Omron CX-Programmer project NewProject (CX-Programmer 9.75)

# PLC parkir: CP1E N20

## Global symbols (name address type ; comment)
0.00 BOOL  ; MULAI
0.01 BOOL  ; STOP
0.02 BOOL  ; SENSOR MASUK
0.03 BOOL  ; SENSOR KELUAR
0.04 BOOL  ; RESET
100.00 BOOL  ; Portal Masuk
100.01 BOOL  ; Portal Keluar
100.02 BOOL  ; SPACE
100.03 BOOL  ; FULL
100.04 BOOL  ; FULL
10.00 BOOL  ; Relay
C2 CHANNEL  ; CNTR
T000 BOOL  ; TIMER
T001 BOOL  ; TIMER

## Program NewProgram1 (cyclic task 0)

### Section Section1

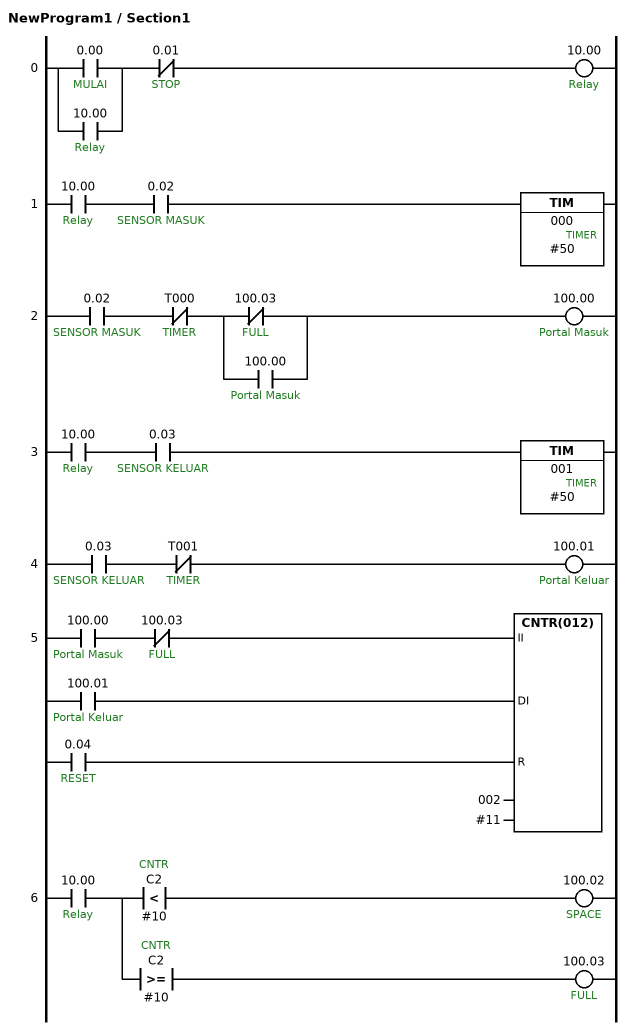
; rung 0
LD 0.00  ; MULAI
OR 10.00  ; Relay
ANDNOT 0.01  ; STOP
OUT 10.00  ; Relay
; rung 1
LD 10.00  ; Relay
AND 0.02  ; SENSOR MASUK
TIM 000 #50  ; TIMER
; rung 2
LD 0.02  ; SENSOR MASUK
ANDNOT T000  ; TIMER
LDNOT 100.03  ; FULL
OR 100.00  ; Portal Masuk
ANDLD
OUT 100.00  ; Portal Masuk
; rung 3
LD 10.00  ; Relay
AND 0.03  ; SENSOR KELUAR
TIM 001 #50  ; TIMER
; rung 4
LD 0.03  ; SENSOR KELUAR
ANDNOT T001  ; TIMER
OUT 100.01  ; Portal Keluar
; rung 5
LD 100.00  ; Portal Masuk
ANDNOT 100.03  ; FULL
LD 100.01  ; Portal Keluar
LD 0.04  ; RESET
CNTR(012) 002 #11
; rung 6
LD 10.00  ; Relay
OUT TR0
AND<(310) C2 #10  ; CNTR
OUT 100.02  ; SPACE
LD TR0
AND>=(325) C2 #10  ; CNTR
OUT 100.03  ; FULL

### Section END
; rung 0
END(001)